Staubli VAL3: onF8Event.pgx

program onF8Event()
  local bool l_bUndo
  local string l_sNew
  local string l_sString
  local num l_nResult
begin
  // look if the bButton is enable
  if bButton[7]
    //
    // new
    //
    call alreadyExist(l_sNew,l_bUndo)
    if !l_bUndo and l_sNew!=""
      call prog:new(l_sNew,l_nResult)
      if l_nResult==0
        logMsg("[KERNEL] INTERFACE:Create the new program: "+l_sNew)
        sEvent=l_sNew
        call buildList()
      else
        popUpMsg("error code: "+toString("",l_nResult))
        logMsg("[KERNEL] INTERFACE:Create the new program: "+l_sNew+" error code "+toString("",l_nResult))
      endIf
    endIf
  endIf
end
